{attribute 'GeneratedUsingTerminal: AX8118-0100-0102-0102'}
{attribute addProperty BoxType "AX8118-0100-0102-0102"}
{attribute addProperty Id "DeviceDevice_6E2575772Device_SafetyDevice_Safety_C21945A160Ch_ACh_A_D18C6F1622WcStateAT %I*WcState_B516A2644InfoDataAT %I*InfoData_D1E293FD11"}
{attribute addProperty CRC "394541365"}
{attribute addProperty Size "99"}
TYPE AX8118_17843935 EXTENDS EtcSlaveTerminalBase_947E5A46 :
STRUCT
	{attribute addProperty Name "Device"}
	Device : Device_6E257577;
	{attribute addProperty Name "Device_Safety"}
	Device_Safety : Device_Safety_C21945A1;
	{attribute addProperty Name "Ch_A"}
	Ch_A : Ch_A_D18C6F16;
	{attribute addProperty Name "WcState"}
	WcState : WcState_B516A264;
	{attribute addProperty Name "InfoData"}
	InfoData : InfoData_D1E293FD;
END_STRUCT
END_TYPE

(* stored: Version 1.2.0.0, ProductVersion 3.1.4024.9
   DUT AX8118_17843935: Id {005d0eb3-6a28-49f4-9d64-151c7b16337b} *)
